// TIA Portal V18 program export: 1 tag tables, 0 data types, 0 data blocks, 1 code blocks (in call order from the OBs), 0 instance data blocks

VAR_GLOBAL   // PLC tag table "默认变量表"
   Tag_1 AT %M0.0 : Bool;
   Tag_2 AT %M0.1 : Bool;
   Tag_3 AT %M0.2 : Bool;
   Tag_4 AT %M0.3 : Bool;
END_VAR

ORGANIZATION_BLOCK "Main"   // OB1, LAD, ProgramCycle
TITLE = "Main Program Sweep (Cycle)"
{ S7_Optimized_Access := 'TRUE' }
VERSION : 0.1
// stored: AutoNumber true, IsIECCheckEnabled false, SetENOAutomatically false
BEGIN

REGION Network 1
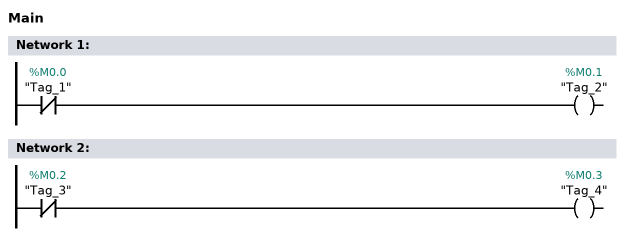
   RUNG wire#powerrail
      I_Contact( "Tag_1" )
      Coil( "Tag_2" )
   END_RUNG
   // the same network as SCL:
   "Tag_2" := NOT "Tag_1";
END_REGION

REGION Network 2
   RUNG wire#powerrail
      I_Contact( "Tag_3" )
      Coil( "Tag_4" )
   END_RUNG
   // the same network as SCL:
   "Tag_4" := NOT "Tag_3";
END_REGION
END_ORGANIZATION_BLOCK
